{attribute 'qualified_only'}
VAR_GLOBAL
	nTemp AT %I*: INT;
END_VAR

(* stored: Version 1.1.0.1, ProductVersion 3.1.4024.12
   GVL GVL_Thermocouple: Id {4a822a92-2427-4cfe-94a6-e1e6615faab7} *)
